METHOD Execute : HRESULT
VAR_INST
	_GetEventState	: UINT; // Step variable
	_BufferOverflow : BOOL; // Buffer maximum reached
END_VAR

VAR
	_TmpAlarm : Tc3_PackML_V2.ST_Alarm; // temp. Alarm structure
	_hr		  : HRESULT;				// HResult
END_VAR
IF __ISVALIDREF(_AdminTag) THEN
	IF _InternalErrorAck AND _InternalError THEN
		_InternalError := FALSE;
	END_IF

	IF _InternalError THEN
		RETURN;
	END_IF

	IF THIS^.GetTimeZone THEN
		IF THIS^.TimeZone() THEN
			THIS^.GetTimeZone := FALSE;
		END_IF
	END_IF

	IF NOT THIS^.GetTimeZone AND THIS^.EventsSubscribed THEN
		Execute := SUPER^.Execute(); // retrieve events
		CASE _GetEventState OF
			0: // Idle
				IF CntAlarmsRaised > 0 THEN
					THIS^.NewEvent := FALSE;
					_GetEventState := _GetEventState + 1;
				END_IF

			1: // handle the event		
				IF aEventInfoBuffer[CntAlarmsRaised].fbRequestEventText.bError THEN
					Tc2_System.ADSLOGSTR(msgCtrlMask := cMsgCtrlMask, msgFmtStr := Tc2_Standard.CONCAT(cBaseMsg, 'Execute: %s'), strArg := 'REQUEST EVENTTEXT ERROR');
					_GetEventState := 0;
					_InternalError := TRUE;
				ELSIF NOT aEventInfoBuffer[CntAlarmsRaised].fbRequestEventText.bBusy THEN
					aEventInfoBuffer[CntAlarmsRaised].fbRequestEventText.GetString(aEventInfoBuffer[CntAlarmsRaised].EventText, SIZEOF(Tc3_PackML_V2.ST_Alarm.Message));
					_hr := THIS^.WriteAlarmTags(Alarm_Ref	  := _TmpAlarm,
												EventInfo_Ref := THIS^.aEventInfoBuffer[CntAlarmsRaised],
												Trigger		  := TRUE,
												AlarmIndex	  := CntAlarmsRaised);

					IF Tc3_Module.SUCCEEDED(_hr) THEN
						// Critical / StopReason 
						IF THIS^.aEventInfoBuffer[CntAlarmsRaised].eSeverity = TcEventSeverity.Critical THEN // Check "Critical" --> Stop reason
							_hr := THIS^.AlarmArrayHandler(NewAlarm_Ref			:= _TmpAlarm,
														   ActAlarmsCounter_Ref := UnclearedStopReasons,
														   MaxArrayElements		:= Tc3_PackML_V2.MaxStopReasons,
														   pAlarmArray			:= ADR(_AdminTag.StopReason),
														   BufferOverflow_Ref	:= _BufferOverflow);

							IF _BufferOverflow THEN
								Tc2_System.ADSLOGSTR(msgCtrlMask := Tc2_System.ADSLOG_MSGTYPE_ERROR, msgFmtStr := Tc2_Standard.CONCAT(cBaseMsg, 'Execute: %s'), strArg := 'Stop reason Buffer is full / FIFO active');
								_BufferOverflow := FALSE;
							END_IF

						// Alarm (StopReason) 
						ELSIF THIS^.aEventInfoBuffer[CntAlarmsRaised].eSeverity = TcEventSeverity.Error THEN // Check "Error" --> Alarm

							// Alarm handling
							_hr := THIS^.AlarmArrayHandler(NewAlarm_Ref			:= _TmpAlarm,
														   ActAlarmsCounter_Ref := UnclearedAlarms,
														   MaxArrayElements		:= Tc3_PackML_V2.MaxAlarms,
														   pAlarmArray			:= ADR(_AdminTag.Alarm),
														   BufferOverflow_Ref	:= _BufferOverflow);

							IF _BufferOverflow THEN
								Tc2_System.ADSLOGSTR(msgCtrlMask := Tc2_System.ADSLOG_MSGTYPE_ERROR, msgFmtStr := Tc2_Standard.CONCAT(cBaseMsg, 'Execute: %s'), strArg := 'Alarm Buffer is full / FIFO active');
								_BufferOverflow := FALSE;
							END_IF

							// to StopReason
							IF _AlarmToStopReason AND Tc3_Module.SUCCEEDED(_hr) THEN
								_hr := THIS^.AlarmArrayHandler(NewAlarm_Ref			:= _TmpAlarm,
															   ActAlarmsCounter_Ref := UnclearedStopReasons,
															   MaxArrayElements		:= Tc3_PackML_V2.MaxStopReasons,
															   pAlarmArray			:= ADR(_AdminTag.StopReason),
															   BufferOverflow_Ref	:= _BufferOverflow);

								IF _BufferOverflow THEN
									Tc2_System.ADSLOGSTR(msgCtrlMask := Tc2_System.ADSLOG_MSGTYPE_ERROR, msgFmtStr := Tc2_Standard.CONCAT(cBaseMsg, 'Execute: %s'), strArg := 'Stop reason Buffer is full / FIFO active');
									_BufferOverflow := FALSE;
								END_IF
							END_IF
						// Warning (StopReason) 
						ELSIF THIS^.aEventInfoBuffer[CntAlarmsRaised].eSeverity = TcEventSeverity.Warning THEN // Check "Warning" --> Warning
							_hr := THIS^.AlarmArrayHandler(NewAlarm_Ref			:= _TmpAlarm,
														   ActAlarmsCounter_Ref := UnclearedWarnings,
														   MaxArrayElements		:= Tc3_PackML_V2.MaxWarnings,
														   pAlarmArray			:= ADR(_AdminTag.Warning),
														   BufferOverflow_Ref	:= _BufferOverflow);

							IF _BufferOverflow THEN
								Tc2_System.ADSLOGSTR(msgCtrlMask := Tc2_System.ADSLOG_MSGTYPE_ERROR, msgFmtStr := Tc2_Standard.CONCAT(cBaseMsg, 'Execute: %s'), strArg := 'Warning Buffer is full / FIFO active');
								_BufferOverflow := FALSE;
							END_IF

							// to StopReason
							IF _WarningToStopReason AND Tc3_Module.SUCCEEDED(_hr) THEN
								_hr := THIS^.AlarmArrayHandler(NewAlarm_Ref			:= _TmpAlarm,
															   ActAlarmsCounter_Ref := UnclearedStopReasons,
															   MaxArrayElements		:= Tc3_PackML_V2.MaxStopReasons,
															   pAlarmArray			:= ADR(_AdminTag.StopReason),
															   BufferOverflow_Ref	:= _BufferOverflow);

								IF _BufferOverflow THEN
									Tc2_System.ADSLOGSTR(msgCtrlMask := Tc2_System.ADSLOG_MSGTYPE_ERROR, msgFmtStr := Tc2_Standard.CONCAT(cBaseMsg, 'Execute: %s'), strArg := 'Stop reason Buffer is full / FIFO active');
									_BufferOverflow := FALSE;
								END_IF
							END_IF
						END_IF

						IF Tc3_Module.SUCCEEDED(_hr) THEN
							CntAlarmsRaised := CntAlarmsRaised - 1;
							_GetEventState	:= 0;
						END_IF
					END_IF
				END_IF

		ELSE
			Tc2_System.ADSLOGSTR(msgCtrlMask := cMsgCtrlMask, msgFmtStr := Tc2_Standard.CONCAT(cBaseMsg, 'Execute: %s'), strArg := 'Case Idx error');
			_InternalError := TRUE;
		END_CASE

		THIS^.GetMsgInfos();
	END_IF
ELSE
	IF NOT _InternalError THEN
		// Set internal Error
		Tc2_System.ADSLOGSTR(msgCtrlMask := cMsgCtrlMask, msgFmtStr := Tc2_Standard.CONCAT(cBaseMsg, 'Execute: %s'), strArg := 'Input-reference error');
		_InternalError := TRUE;
	END_IF
END_IF
END_METHOD

METHOD PUBLIC GetMsgInfos : ST_PackML_aEventInfo
VAR
	_Iterator : DINT; // FOR-Loop iterator						
END_VAR
// StopReason

// Reset
GetMsgInfos.StopReason.Active		   := FALSE;
GetMsgInfos.StopReason.NumberActive	   := 0;
GetMsgInfos.StopReason.NumberConfirmed := 0;
GetMsgInfos.StopReason.NumberCleared   := 0;
FOR _Iterator := 1 TO Tc3_PackML_V2.MaxStopReasons DO
	// Active
	IF _AdminTag.StopReason[_Iterator].Trigger THEN
		GetMsgInfos.StopReason.Active		:= TRUE;
		GetMsgInfos.StopReason.NumberActive := GetMsgInfos.StopReason.NumberActive + 1;
	END_IF

	// Confirmed
	IF NOT _AdminTag.StopReason[_Iterator].Trigger AND (_AdminTag.StopReason[_Iterator].Category = 4) THEN
		GetMsgInfos.StopReason.NumberConfirmed := GetMsgInfos.StopReason.NumberConfirmed + 1;
	END_IF
END_FOR

// Alarm		

// Reset
GetMsgInfos.Alarm.Active		  := FALSE;
GetMsgInfos.Alarm.NumberActive	  := 0;
GetMsgInfos.Alarm.NumberConfirmed := 0;
GetMsgInfos.Alarm.NumberCleared	  := 0;
FOR _Iterator := 1 TO Tc3_PackML_V2.MaxAlarms DO
	// Active
	IF _AdminTag.Alarm[_Iterator].Trigger THEN
		GetMsgInfos.Alarm.Active	   := TRUE;
		GetMsgInfos.Alarm.NumberActive := GetMsgInfos.StopReason.NumberActive + 1;
	END_IF

	// Confirmed
	IF NOT _AdminTag.Alarm[_Iterator].Trigger AND (_AdminTag.Alarm[_Iterator].Category = 3) THEN
		GetMsgInfos.Alarm.NumberConfirmed := GetMsgInfos.Alarm.NumberConfirmed + 1;
	END_IF
END_FOR

// Warning		

// Reset
GetMsgInfos.Warning.Active			:= FALSE;
GetMsgInfos.Warning.NumberActive	:= 0;
GetMsgInfos.Warning.NumberConfirmed := 0;
GetMsgInfos.Warning.NumberCleared	:= 0;
FOR _Iterator := 1 TO Tc3_PackML_V2.MaxWarnings DO
	// Active
	IF _AdminTag.Warning[_Iterator].Trigger THEN
		GetMsgInfos.Warning.Active		 := TRUE;
		GetMsgInfos.Warning.NumberActive := GetMsgInfos.StopReason.NumberActive + 1;
	END_IF

	// Confirmed
	IF NOT _AdminTag.Warning[_Iterator].Trigger AND (_AdminTag.Warning[_Iterator].Category = 2) THEN
		GetMsgInfos.Warning.NumberConfirmed := GetMsgInfos.Warning.NumberConfirmed + 1;
	END_IF
END_FOR

// Cleared --> historizied
GetMsgInfos.HistorizedMsg := TO_UDINT(MsgInHistory);
FOR _Iterator := 1 TO Tc3_PackML_V2.MaxHistoryAlarms DO
	IF (_AdminTag.AlarmHistory[_Iterator].Category = 4) THEN // StopReason
		GetMsgInfos.StopReason.NumberCleared := GetMsgInfos.StopReason.NumberCleared + 1;
	ELSIF (_AdminTag.AlarmHistory[_Iterator].Category = 3) THEN // Alarm
		GetMsgInfos.Alarm.NumberCleared := GetMsgInfos.Alarm.NumberCleared + 1;
	ELSIF (_AdminTag.AlarmHistory[_Iterator].Category = 2) THEN // Warning
		GetMsgInfos.Warning.NumberCleared := GetMsgInfos.Warning.NumberCleared + 1;
	END_IF

	IF (_AdminTag.AlarmHistory[_Iterator].Category = 0) THEN
		EXIT;
	END_IF
END_FOR
END_METHOD

PROPERTY InitComplete : BOOL
GET
InitComplete := _InitComplete;
END_GET
END_PROPERTY

METHOD Initialize : BOOL
IF NOT EventsSubscribed THEN
	EventListener(Subscribe := TRUE, Subscribed => EventsSubscribed);
END_IF

Initialize := EventsSubscribed;
END_METHOD

PROPERTY InSimulation : BOOL
GET
InSimulation := _InSimulation;
END_GET
SET
_InSimulation := InSimulation;
END_SET
END_PROPERTY

PROPERTY InternalErrorAck : BOOL
GET
InternalErrorAck := _InternalErrorAck;
END_GET
SET
_InternalErrorAck := InternalErrorAck;
END_SET
END_PROPERTY

METHOD PRIVATE MoveAlarmToHistory : HRESULT
VAR_INPUT
	pAlarmArray		 : POINTER TO ST_Alarm; // Pointer to Array of ST_Alarm of Alarm / Warning / Stop reason
	ActAlarms_Ref	 : REFERENCE TO DINT;	// Reference to couter of active Alarm / Warning / Stop reason
	MaxArrayElements : INT;					// max. Alarm / Warning / Stop reason constant
	EventId			 : UDINT;				// EventId of Alarm / Warning / Stop reason to confirm
	Timestamp		 : ULINT;				// Event Timestamp
END_VAR

VAR
	_Iterator				  : INT;					// FOR-Loop iterator	
	_Iterator2				  : DINT;					// FOR-Loop iterator	
	_TempTimestruct			  : TIMESTRUCT;				// TimeStruct for ACK Time
	_TmpAlarm				  : Tc3_PackML_V2.ST_Alarm; // temp. Alarm Structure
	_hr						  : HRESULT;				// hresult
	_MaxArrayElementsInternal : INT;					// calculated internal Array upper border
	_BufferOverflow			  : BOOL;					// Buffer maximum reached
END_VAR
IF __ISVALIDREF(ActAlarms_Ref) THEN
	_MaxArrayElementsInternal := (MaxArrayElements - 1);

	// Search Alarm in Array
	FOR _Iterator := 0 TO _MaxArrayElementsInternal DO
		IF (pAlarmArray[_Iterator].ID = TO_DINT(EventId)) THEN
			// TimeZone
			THIS^.fbSpecificLocalTime(in := Tc2_Utilities.FILETIME64_TO_SYSTEMTIME(Timestamp), tzInfo := fbTimeZone.tzInfo, out => _TempTimestruct);

			// Copy Alarm to local Memory
			Tc2_System.MEMCPY(destAddr := ADR(_TmpAlarm), srcAddr := ADR(pAlarmArray[_Iterator]), n := SIZEOF(Tc3_PackML_V2.ST_Alarm));

			// Set ACK Timestamp	
			_TmpAlarm.AckDateTime[0] := TO_DINT(_TempTimestruct.wYear);
			_TmpAlarm.AckDateTime[1] := TO_DINT(_TempTimestruct.wMonth);
			_TmpAlarm.AckDateTime[2] := TO_DINT(_TempTimestruct.wDay);
			_TmpAlarm.AckDateTime[3] := TO_DINT(_TempTimestruct.wHour);
			_TmpAlarm.AckDateTime[4] := TO_DINT(_TempTimestruct.wMinute);
			_TmpAlarm.AckDateTime[5] := TO_DINT(_TempTimestruct.wSecond);
			_TmpAlarm.AckDateTime[6] := TO_DINT(_TempTimestruct.wMilliseconds);
			_TmpAlarm.Trigger		 := FALSE;

			// Move to History	
			_hr := THIS^.AlarmArrayHandler(NewAlarm_Ref			:= _TmpAlarm,
										   ActAlarmsCounter_Ref := THIS^.MsgInHistory,
										   MaxArrayElements		:= Tc3_PackML_V2.MaxHistoryAlarms,
										   pAlarmArray			:= ADR(_AdminTag.AlarmHistory),
										   BufferOverflow_Ref	:= _BufferOverflow);

			IF _BufferOverflow THEN
				Tc2_System.ADSLOGSTR(msgCtrlMask := Tc2_System.ADSLOG_MSGTYPE_ERROR, msgFmtStr := Tc2_Standard.CONCAT(cBaseMsg, 'MoveAlarmToHistory: %s'), strArg := 'History Buffer is full / FIFO active');
			END_IF

			IF Tc3_Module.SUCCEEDED(_hr) THEN
				// Close empty entry in source array
				Tc2_System.MEMMOVE(destAddr := ADR(pAlarmArray[_Iterator]), srcAddr := ADR(pAlarmArray[_Iterator + 1]), n := (SIZEOF(Tc3_PackML_V2.ST_Alarm) * (TO_UINT((_MaxArrayElementsInternal) - (_Iterator))))); // move Alarm 
				Tc2_System.MEMSET(destAddr := ADR(pAlarmArray[_MaxArrayElementsInternal]), fillByte := 0, n := SIZEOF(Tc3_PackML_V2.ST_Alarm));																		   // delete last entry

				// Find next empty entry index 
				FOR _Iterator2 := 0 TO (_MaxArrayElementsInternal) DO
					IF (pAlarmArray[_Iterator2].Message = '') OR (_Iterator2 = _MaxArrayElementsInternal) THEN
						IF _Iterator2 > 0 THEN
							ActAlarms_Ref := _Iterator2 - 1;
						ELSE
							ActAlarms_Ref := _Iterator2;
						END_IF

						EXIT;
					END_IF
				END_FOR
			END_IF

			EXIT;
		END_IF
	END_FOR

	MoveAlarmToHistory := S_OK;
ELSE
	// Set internal Error
	Tc2_System.ADSLOGSTR(msgCtrlMask := cMsgCtrlMask, msgFmtStr := Tc2_Standard.CONCAT(cBaseMsg, 'MoveAlarmToHistory: %s'), strArg := 'Input-reference error');
	MoveAlarmToHistory := E_FAIL;
	_InternalError	   := TRUE;
END_IF
END_METHOD

PROPERTY Name : STRING
GET
END_GET
SET
_Name := Name;
END_SET
END_PROPERTY

METHOD OnAlarmCleared : HRESULT
VAR_INPUT
	fbEvent : REFERENCE TO FB_TcEvent; // Reference to FB_Event (Callback!)
END_VAR

VAR_INST
	_idxEventReceived : INT; // Event index
END_VAR

VAR
	_hr : HRESULT; // hresult
END_VAR
// Move Alarm to History
IF fbEvent.eSeverity = TcEventSeverity.Critical THEN // Check "Critical" --> Stop reason
	_hr := MoveAlarmToHistory(MaxArrayElements := Tc3_PackML_V2.MaxStopReasons,
							  EventId		   := fbEvent.nEventId,
							  pAlarmArray	   := ADR(_AdminTag.StopReason),
							  Timestamp		   := fbEvent.nTimestamp,
							  ActAlarms_Ref	   := UnclearedStopReasons);
ELSIF fbEvent.eSeverity = TcEventSeverity.Error THEN // Check "Error" --> Alarm
	_hr := MoveAlarmToHistory(MaxArrayElements := Tc3_PackML_V2.MaxAlarms,
							  EventId		   := fbEvent.nEventId,
							  pAlarmArray	   := ADR(_AdminTag.Alarm),
							  Timestamp		   := fbEvent.nTimestamp,
							  ActAlarms_Ref	   := UnclearedAlarms);

	IF _AlarmToStopReason AND Tc3_Module.SUCCEEDED(_hr) THEN
		_hr := THIS^.ClearStopReason(pAlarmArray	  := ADR(_AdminTag.StopReason),
									 ActAlarms_Ref	  := THIS^.UnclearedStopReasons,
									 MaxArrayElements := Tc3_PackML_V2.MaxStopReasons,
									 EventId		  := fbEvent.nEventId);
	END_IF
ELSIF fbEvent.eSeverity = TcEventSeverity.Warning THEN // Check "Warning" --> Warning
	_hr := MoveAlarmToHistory(MaxArrayElements := Tc3_PackML_V2.MaxWarnings,
							  EventId		   := fbEvent.nEventId,
							  pAlarmArray	   := ADR(_AdminTag.Warning),
							  Timestamp		   := fbEvent.nTimestamp,
							  ActAlarms_Ref	   := UnclearedWarnings);

	IF _WarningToStopReason AND Tc3_Module.SUCCEEDED(_hr) THEN
		_hr := THIS^.ClearStopReason(pAlarmArray	  := ADR(_AdminTag.StopReason),
									 ActAlarms_Ref	  := THIS^.UnclearedStopReasons,
									 MaxArrayElements := Tc3_PackML_V2.MaxStopReasons,
									 EventId		  := fbEvent.nEventId);
	END_IF
END_IF

OnAlarmCleared := S_OK; // in order to receive more callbacks (Set <> S_OK in order to cancel the callbacks for this program cycle.)
END_METHOD

// Callback Method
METHOD OnAlarmConfirmed : HRESULT
VAR_INPUT
	fbEvent : REFERENCE TO FB_TcEvent; // Reference to FB_Event (Callback!)
END_VAR

VAR
	_hr : HRESULT; // hresult
END_VAR
// Move Alarm to History
IF __ISVALIDREF(fbEvent) THEN
	// Set ACK Timestamp
	IF fbEvent.eSeverity = TcEventSeverity.Critical THEN // Check "Critical" --> Stop reason
		_hr := ConfirmAlarm(MaxArrayElements := Tc3_PackML_V2.MaxStopReasons,
							EventId			 := fbEvent.nEventId,
							pAlarmArray		 := ADR(_AdminTag.StopReason),
							Timestamp		 := fbEvent.nTimestamp,
							ActAlarms_Ref	 := UnclearedStopReasons);
	ELSIF fbEvent.eSeverity = TcEventSeverity.Error THEN // Check "Error" --> Alarm
		_hr := ConfirmAlarm(MaxArrayElements := Tc3_PackML_V2.MaxAlarms,
							EventId			 := fbEvent.nEventId,
							pAlarmArray		 := ADR(_AdminTag.Alarm),
							Timestamp		 := fbEvent.nTimestamp,
							ActAlarms_Ref	 := UnclearedAlarms);
	ELSIF fbEvent.eSeverity = TcEventSeverity.Warning THEN // Check "Warning" --> Warning
		_hr := ConfirmAlarm(MaxArrayElements := Tc3_PackML_V2.MaxWarnings,
							EventId			 := fbEvent.nEventId,
							pAlarmArray		 := ADR(_AdminTag.Warning),
							Timestamp		 := fbEvent.nTimestamp,
							ActAlarms_Ref	 := UnclearedWarnings);
	END_IF

	OnAlarmConfirmed := S_OK; // in order to receive more callbacks (Set <> S_OK in order to cancel the callbacks for this program cycle.)
ELSE
	// Set internal Error
	Tc2_System.ADSLOGSTR(msgCtrlMask := cMsgCtrlMask, msgFmtStr := Tc2_Standard.CONCAT(cBaseMsg, 'OnAlarmConfirmed: %s'), strArg := 'Input-reference error');
	OnAlarmConfirmed := E_FAIL;
	_InternalError	 := TRUE;
END_IF
END_METHOD

// Callback Method
METHOD OnAlarmRaised : HRESULT
VAR_INPUT
	fbEvent : REFERENCE TO FB_TcEvent; // Reference to FB_Event (Callback!)
END_VAR

VAR
	_TempTimestruct : TIMESTRUCT; // TimeStruct for ACK Time
END_VAR
// when (new) event is triggered -> trigger within cyclic method 'execute'
THIS^.NewEvent := TRUE;

// for local event -> raise counter
CntAlarmsRaised := CntAlarmsRaised + 1;

// save eventinfo locally
THIS^.stEventInfo.Source	  := fbEvent.ipSourceInfo.sName;
THIS^.stEventInfo.eSeverity	  := fbEvent.eSeverity;
THIS^.stEventInfo.EventClass  := fbEvent.EventClass;
THIS^.stEventInfo.EventId	  := fbEvent.nEventId;
THIS^.stEventInfo.ipArguments := fbEvent.ipArguments;

// TimeZone
fbSpecificLocalTime(in := Tc2_Utilities.FILETIME64_TO_SYSTEMTIME(fbEvent.nTimestamp), tzInfo := fbTimeZone.tzInfo, out => _TempTimestruct);

// Timestamp	
THIS^.stEventInfo.TimeRaised[0] := TO_DINT(_TempTimestruct.wYear);
THIS^.stEventInfo.TimeRaised[1] := TO_DINT(_TempTimestruct.wMonth);
THIS^.stEventInfo.TimeRaised[2] := TO_DINT(_TempTimestruct.wDay);
THIS^.stEventInfo.TimeRaised[3] := TO_DINT(_TempTimestruct.wHour);
THIS^.stEventInfo.TimeRaised[4] := TO_DINT(_TempTimestruct.wMinute);
THIS^.stEventInfo.TimeRaised[5] := TO_DINT(_TempTimestruct.wSecond);
THIS^.stEventInfo.TimeRaised[6] := TO_DINT(_TempTimestruct.wMilliseconds);
Tc2_System.MEMSET(destAddr := ADR(stEventInfo.TimeCleared), fillByte := 0, n := SIZEOF(stEventInfo.TimeCleared));
Tc2_System.MEMSET(destAddr := ADR(stEventInfo.TimeConfirmed), fillByte := 0, n := SIZEOF(stEventInfo.TimeConfirmed));

// store event info globally
aEventInfoBuffer[CntAlarmsRaised] := stEventInfo;

// activate requests in event triggered method 'OnMessageSent' to get related request info
aEventInfoBuffer[CntAlarmsRaised].fbRequestEventText.Request(eventClass := aEventInfoBuffer[CntAlarmsRaised].EventClass,
															 nEventId	:= aEventInfoBuffer[CntAlarmsRaised].EventId,
															 nLangId	:= 1033,
															 ipArgs		:= aEventInfoBuffer[CntAlarmsRaised].ipArguments);

OnAlarmRaised := S_OK; // in order to receive more callbacks (Set <> S_OK in order to cancel the callbacks for this program cycle.)
END_METHOD

PROPERTY ParentResponseDefinitions : ARRAY[0..4] OF SPT_BaseTypes.E_AlarmResponse
GET
ParentResponseDefinitions := _ParentResponseDefinitions;
END_GET
SET
_ParentResponseDefinitions := ParentResponseDefinitions;
END_SET
END_PROPERTY

METHOD Reset : BOOL
// This may or may not be called depending on the component type 

// which derives FB_ComponentBase
F_ClearAllEventsInClass(PackMLEventHandlerAlarms);
Reset := TRUE;
END_METHOD

METHOD PUBLIC TimeZone : BOOL
VAR_INST
	_Step : USINT; // Step Variable
END_VAR
CASE _Step OF
	0: // Start to get local Timezone 
		fbTimeZone.bExecute := TRUE;
		IF fbTimeZone.bBusy THEN
			_Step := _Step + 1;
		END_IF

	1: // set 
		fbTimeZone.bExecute := FALSE;
		_Step				:= 0;
		TimeZone			:= TRUE;

ELSE
	Tc2_System.ADSLOGSTR(msgCtrlMask := cMsgCtrlMask, msgFmtStr := Tc2_Standard.CONCAT(cBaseMsg, 'TimeZone: %s'), strArg := 'Case Idx error');
	_InternalError := TRUE;
END_CASE

fbTimeZone(sNetID := '');
IF fbTimeZone.bError THEN
	Tc2_System.ADSLOGSTR(msgCtrlMask := cMsgCtrlMask, msgFmtStr := Tc2_Standard.CONCAT(cBaseMsg, 'fbTimeZone ErrID: %s'), strArg := TO_STRING(fbTimeZone.nErrID));
	_InternalError := TRUE;
END_IF
END_METHOD

PROPERTY WarningToStopReason : BOOL
SET
_WarningToStopReason := WarningToStopReason;
END_SET
END_PROPERTY

METHOD PRIVATE WriteAlarmTags : HRESULT;
VAR_INPUT
	Alarm_Ref	  : REFERENCE TO Tc3_PackML_V2.ST_Alarm; // Reference to ST_Alarm of an new Alarm / Warning / Stop reason
	EventInfo_Ref : REFERENCE TO ST_EventInfo;			 // Reference to ST_EventInfo
	Trigger		  : BOOL;								 // Set / Reset Trigger in PML Structure
	AlarmIndex	  : DINT;								 // Alarm index
END_VAR
IF __ISVALIDREF(Alarm_Ref) AND __ISVALIDREF(EventInfo_Ref) THEN
	Alarm_Ref.ID	   := TO_DINT(EventInfo_Ref.EventId);
	Alarm_Ref.Value	   := AlarmIndex;
	Alarm_Ref.Message  := EventInfo_Ref.EventText;
	Alarm_Ref.Category := TO_DINT(EventInfo_Ref.eSeverity); // Verbose:=0, Info:=1, Warning:=2, Error:=3, Critical:=4
	Alarm_Ref.Trigger  := Trigger;
	Alarm_Ref.DateTime := EventInfo_Ref.TimeRaised;
	WriteAlarmTags	   := S_OK;
ELSE
	// Set internal Error
	Tc2_System.ADSLOGSTR(msgCtrlMask := cMsgCtrlMask, msgFmtStr := Tc2_Standard.CONCAT(cBaseMsg, 'WriteAlarmTags: %s'), strArg := 'Input-reference error');
	WriteAlarmTags := E_FAIL;
	_InternalError := TRUE;
END_IF
END_METHOD

END_FUNCTION_BLOCK

// Project Information/F_GetCompany
// This function has been automatically generated from the project information.
{attribute 'signature_flag' := '1073741824'}
{attribute 'TcGenerated'}
{attribute 'no-analysis'}
FUNCTION F_GetCompany : WSTRING
VAR_INPUT
	
END_VAR

F_GetCompany := "Beckhoff Automation LLC";

END_FUNCTION

// Project Information/F_GetTitle
// This function has been automatically generated from the project information.
{attribute 'signature_flag' := '1073741824'}
{attribute 'TcGenerated'}
{attribute 'no-analysis'}
FUNCTION F_GetTitle : WSTRING
VAR_INPUT
	
END_VAR

F_GetTitle := "SPT Components";

END_FUNCTION

// Project Information/F_GetVersion
// This function has been automatically generated from the project information.
{attribute 'signature_flag' := '1073741824'}
{attribute 'TcGenerated'}
{attribute 'no-analysis'}
FUNCTION F_GetVersion : ST_LibVersion
VAR_INPUT
	
END_VAR

F_GetVersion.iMajor := 3;
F_GetVersion.iMinor := 9;
F_GetVersion.iBuild := 0;
F_GetVersion.iRevision := 0;
F_GetVersion.sVersion := '3.9.0';
F_GetVersion.nFlags := 1;

END_FUNCTION

// Sensors/FB_DigitalSensor
FUNCTION_BLOCK FB_DigitalSensor EXTENDS FB_ComponentBase IMPLEMENTS I_DigitalSensorBase
VAR
	HardwareInput AT %I*		: BOOL;			  // Hardware input bit from the physical sensor
	_DebounceMode				: E_DebounceMode; // Defines the debounce model that will filter the sensor's output to the program
	_DebounceTime				: TIME;			  // Time input parameter for use in Debounce functionality
	_Inverted					: BOOL;			  // Defines the output polarity of the sensor - a "TRUE" value will result in the signal of the sensor being inverted
	_SimulationInput			: BOOL;			  // Provides configuration input to the simulation functionality
	_SimulationTimebase			: UDINT;
	_SimulationMode				: E_SensorSimulationMode; // Defines the mode of operation for the simulation functionality of this component
	_TimeActive					: TIME;					  // Tracks the amount of time that the sensor has been in an active state
	_TimeInactive				: TIME;					  // Tracks the amount of time that the sensor has been in an inactive state
	_Active						: BOOL;
	TON_ActiveTimer				: Tc2_Standard.TON; // Tracks the amount of time that the sensor has been in an active state
	TON_InactiveTimer			: Tc2_Standard.TON; // Tracks the amount of time that the sensor has been in an inactive state
	TON_DebounceTimer			: Tc2_Standard.TON; // Utilized in the debounce implementation
	TP_DebounceTimer			: Tc2_Standard.TP;	// Utilized in the debounce implementation
	DigitalSensor_HMI			: ST_DigitalSensor_HMI;
	SimulationPulse1_TP			: Tc2_Standard.TP; // Pulse Timer for simulated sensor pulse generation
	SimulationPulse2_TP			: Tc2_Standard.TP; // Pulse Timer for simulated sensor pulse generation
	HMICommand_DigitalSensor_RT : R_TRIG;
END_VAR

METHOD PUBLIC CyclicLogic
VAR_INPUT
END_VAR
SUPER^.CyclicLogic();
IF _Simulate THEN
	CASE _SimulationMode OF
		E_SensorSimulationMode.InputDriven:
			_Active := _SimulationInput;

		E_SensorSimulationMode.Periodic:
			SimulationPulse1_TP(IN := NOT SimulationPulse2_TP.Q, PT := UDINT_TO_TIME(_SimulationTimebase));
			SimulationPulse2_TP(IN := NOT SimulationPulse1_TP.Q, PT := UDINT_TO_TIME(_SimulationTimebase));
			_Active := SimulationPulse2_TP.Q;
	END_CASE
ELSE
	_Active := ProcessInput(Input := HardwareInput);
END_IF
END_METHOD

PROPERTY Active : BOOL
GET
Active := _Active;
END_GET
END_PROPERTY

PROPERTY DebounceMode : E_DebounceMode
GET
DebounceMode := _DebounceMode;
END_GET
SET
_DebounceMode := DebounceMode;
END_SET
END_PROPERTY

PROPERTY DebounceTime : TIME
GET
DebounceTime := _DebounceTime;
END_GET
SET
_DebounceTime := DebounceTime;
END_SET
END_PROPERTY

PROPERTY Inverted : BOOL
GET
Inverted := _Inverted;
END_GET
SET
_Inverted := Inverted;
END_SET
END_PROPERTY

PROPERTY SimulationInput : BOOL
GET
SimulationInput := _SimulationInput;
END_GET
SET
_SimulationInput := SimulationInput;
END_SET
END_PROPERTY

PROPERTY SimulationMode : E_SensorSimulationMode
GET
SimulationMode := _SimulationMode;
END_GET
SET
_SimulationMode := SimulationMode;
END_SET
END_PROPERTY

PROPERTY SimulationTimeBase : UDINT
GET
SimulationTimeBase := _SimulationTimebase;
END_GET
SET
_SimulationTimeBase := SimulationTimebase;
END_SET
END_PROPERTY

PROPERTY TimeActive : TIME
GET
TimeActive := _TimeActive;
END_GET
END_PROPERTY

PROPERTY TimeInactive : TIME
GET
TimeInactive := _TimeInactive;
END_GET
END_PROPERTY

METHOD PROTECTED HMICommunication
// Extend this method in extended FBs to communicate specific implementation data
SUPER^.HMICommunication();

// Process HMI requests

// Replace 'FALSE' below with further momentary commands (myCommand XOR myOtherCommand XOR...)
HMICommand_DigitalSensor_RT(CLK := (ComponentBase_HMI.Status.HMIControlAvailable AND NOT HMICommandActive_Base) AND (FALSE));

// Signal to FB_ComponentBase that a command is active
HMICommandActive_Descendant := ComponentBase_HMI.Status.HMIControlAvailable AND (DigitalSensor_HMI.Config.DebounceMode <> _DebounceMode OR DigitalSensor_HMI.Config.DebounceTime <> _DebounceTime OR DigitalSensor_HMI.Config.Inverted <> _Inverted OR DigitalSensor_HMI.Config.SimulationMode <> _SimulationMode OR DigitalSensor_HMI.Config.SimulationTimebase <> _SimulationTimebase);

// Process HMI requests
IF HMICommand_DigitalSensor_RT.Q THEN // If a request has been issued by the HMI, and a previous request has not just finished being processed

	//	IF AxisBaseHMI.Command.xxx THEN

	//		Enabled := TRUE;

	//	END_IF
END_IF

IF ComponentBase_HMI.Status.HMIControlAvailable AND NOT HMICommand_DigitalSensor_RT.Q THEN
	IF DigitalSensor_HMI.Config.DebounceMode <> _DebounceMode THEN
		DebounceMode := DigitalSensor_HMI.Config.DebounceMode;
	END_IF

	IF DigitalSensor_HMI.Config.DebounceTime <> _DebounceTime THEN
		DebounceTime := DigitalSensor_HMI.Config.DebounceTime;
	END_IF

	IF DigitalSensor_HMI.Config.Inverted <> _Inverted THEN
		Inverted := DigitalSensor_HMI.Config.Inverted;
	END_IF

	IF DigitalSensor_HMI.Config.SimulationMode <> _SimulationMode THEN
		SimulationMode := DigitalSensor_HMI.Config.SimulationMode;
	END_IF

	IF DigitalSensor_HMI.Config.SimulationTimebase <> _SimulationTimebase THEN
		SimulationTimeBase := DigitalSensor_HMI.Config.SimulationTimebase;
	END_IF
END_IF

// Update HMI status info
DigitalSensor_HMI.Status.Active				:= _Active;
DigitalSensor_HMI.Status.TimeActive			:= TIME_TO_LREAL(_TimeActive) / 1000.0;
DigitalSensor_HMI.Status.TimeInactive		:= TIME_TO_LREAL(_TimeInactive) / 1000.0;
DigitalSensor_HMI.Config.DebounceMode		:= DebounceMode;
DigitalSensor_HMI.Config.DebounceTime		:= DebounceTime;
DigitalSensor_HMI.Config.Inverted			:= Inverted;
DigitalSensor_HMI.Config.SimulationMode		:= SimulationMode;
DigitalSensor_HMI.Config.SimulationTimebase := SimulationTimeBase;
END_METHOD

METHOD PROTECTED Monitoring
SUPER^.Monitoring();

// If flicker counters or other diagnostic systems are desired, their implementation could be here

// Any warnings, errors, or other desired messages would also be generated here

// T#71582M47S295MS is the upper bound of the TIME type, meaning these timers will continue to increase ET for as long as possible
TON_ActiveTimer(IN := _Active, PT := T#71582M47S295MS, ET => _TimeActive);
TON_InactiveTimer(IN := NOT _Active, PT := T#71582M47S295MS, ET => _TimeInactive);
_Busy  := FALSE;
_Error := FALSE;
END_METHOD

METHOD PRIVATE ProcessInput : BOOL
VAR_INPUT
	Input : BOOL;
END_VAR

VAR
	DebouncedInput : BOOL;
END_VAR

VAR_INST
	LastDebouncedInput : BOOL;
	MovingAverage	   : DINT;
END_VAR
CASE DebounceMode OF
	E_DebounceMode.RawInput: // Passes raw input through
		DebouncedInput := Input;

	E_DebounceMode.SimpleFlickerFilter:											 // Requires the raw input to be a consistent value for a set time period before output changes
		TON_DebounceTimer(IN := (Input <> DebouncedInput), PT := _DebounceTime); // runs the timer whenever a differing input is detected
		IF TON_DebounceTimer.Q THEN
			DebouncedInput := Input; // once the raw input has been different for the specified debounce time, the processed input is updated
		END_IF

	E_DebounceMode.EdgeDetectFilter:								   // Updates the processed value immediately on a change from steady state, but mutes any sensor flickers for the specified time immediately following the change
		IF (Input <> DebouncedInput) AND (NOT TP_DebounceTimer.Q) THEN // A differing raw input must be detected outside of the mute window created by the pulse timer
			DebouncedInput := Input;
		END_IF

		TP_DebounceTimer(IN := (DebouncedInput <> LastDebouncedInput), PT := _DebounceTime); // "Q" will be TRUE for tDebounce time after the bProcessedSensorInput value is changed
	E_DebounceMode.MovingAverage:															 // Uses a "moving average"-like calculation to compensate for extremely inconsistent signals - prevents poorly timed flickers from causing disproportionate results
		TON_DebounceTimer(IN := NOT TON_DebounceTimer.Q, PT := T#5MS);						 // Provides a 1ms "polling" trigger
		IF TON_DebounceTimer.Q THEN															 // TRUE once every millisecond
			IF Input THEN																	 // If raw input is currently active at the time of polling
				IF MovingAverage < TIME_TO_DINT(_DebounceTime) THEN							 // If the moving average has not reached its "weight limit" as set by debounce time
					MovingAverage := MovingAverage + 5;										 // Add 1 to the average
				END_IF
			ELSE													 // If raw input is currently inactive at the time of polling
				IF MovingAverage > -TIME_TO_DINT(_DebounceTime) THEN // If the moving average has not reached its "weight limit" as set by debounce time
					MovingAverage := MovingAverage - 5;				 // Subtract 1 from the average
				END_IF
			END_IF
		END_IF

		IF MovingAverage >= 0 THEN
			DebouncedInput := TRUE;
		ELSE
			DebouncedInput := FALSE;
		END_IF
END_CASE

LastDebouncedInput := DebouncedInput; // Update "Last value"
IF _Inverted THEN					  // If signal inversion is requested, invert the signal
	DebouncedInput := NOT DebouncedInput;
END_IF

ProcessInput := DebouncedInput;
END_METHOD

END_FUNCTION_BLOCK

// Sensors/I_DigitalSensorBase
INTERFACE I_DigitalSensorBase

PROPERTY Active : BOOL
GET
END_GET
END_PROPERTY

PROPERTY DebounceMode : E_DebounceMode
GET
END_GET
SET
END_SET
END_PROPERTY

PROPERTY DebounceTime : TIME
GET
END_GET
SET
END_SET
END_PROPERTY

PROPERTY Inverted : BOOL //"High" signal from the sensor will be interpreted as an "inactive" reading when this parameter is TRUE
GET
END_GET
SET
END_SET
END_PROPERTY

PROPERTY SimulationInput : BOOL
GET
END_GET
SET
END_SET
END_PROPERTY

PROPERTY SimulationMode : E_SensorSimulationMode
GET
END_GET
SET
END_SET
END_PROPERTY

PROPERTY TimeActive : TIME
GET
END_GET
END_PROPERTY

PROPERTY TimeInactive : TIME
GET
END_GET
END_PROPERTY

END_INTERFACE

// Solenoids/SolenoidBankBase/FB_SolenoidBankBase
FUNCTION_BLOCK ABSTRACT FB_SolenoidBankBase EXTENDS FB_ComponentBase
VAR
	// Configuration
	Configuration : ARRAY[1..Parameters_Cylinder.MAX_NUMBER_OF_SOLENOIDS] OF ST_SolenoidBankConfig;

	// Counted number of solenoids
	NumberOfSolenoids : UINT;

	// Alarms
	SolenoidBankAlarms : ARRAY[1..SolenoidBankBaseAlarmsCount] OF FB_TcAlarm;
END_VAR

VAR CONSTANT
	SolenoidBankBaseAlarmsCount : UINT := 2;
END_VAR

METHOD PUBLIC AddSolenoid : UINT
VAR_INPUT
	ipCylinder	 : I_Solenoid;
	Number		 : UINT; // This is the number in the IO tree.
	SolenoidType : E_SolenoidType;
END_VAR
IF CheckNumber(Number) AND ipCylinder <> 0 THEN
	NumberOfSolenoids									  := NumberOfSolenoids + 1;
	Configuration[NumberOfSolenoids].ipSolenoid			  := ipCylinder;
	Configuration[NumberOfSolenoids].SolenoidType		  := SolenoidType;
	Configuration[NumberOfSolenoids].SolenoidOutputNumber := Number;
END_IF
END_METHOD

METHOD PRIVATE CheckNumber : BOOL
VAR_INPUT
	Number : UINT;
END_VAR
CheckNumber := TRUE;
IF Number < 1 AND Number > Parameters_Cylinder.MAX_NUMBER_OF_SOLENOIDS THEN
	IF NOT SolenoidBankAlarms[E_CylinderBankAlarms.CylinderNumberOutOfRange].bRaised THEN
		SolenoidBankAlarms[E_CylinderBankAlarms.CylinderNumberOutOfRange].Raise(0);
	END_IF

	CheckNumber := FALSE;
END_IF
END_METHOD

METHOD PROTECTED CreateEvents
SUPER^.CreateEvents();
F_CreateAllEventsInClass(Alarms		:= SolenoidBankAlarms,
						 ClassSize	:= SIZEOF(TC_EVENTS.CylinderBankAlarms),
						 pInitEvent := ADR(TC_EVENTS.CylinderBankAlarms.InitReferenceEvent),
						 Prefix		:= Name);
END_METHOD

// This method serves as the entry point for all underlying FB logic
METHOD PUBLIC CyclicLogic
// This method should be called cyclically by descendant function blocks by invoking SUPER^.CyclicLogic().  Alternatively, the contents of this method could be reimplemented entirely in which case a call to this method would not be necessary.
VAR
	x : UINT;
END_VAR
// Loop through all solenoids that are added.
FOR x := 1 TO NumberOfSolenoids DO
	MapIO(x);
END_FOR
END_METHOD

// Basic component initialization logic
METHOD PROTECTED Initialize : BOOL;
// This method is called by CyclicLogic() as required
VAR
	x : UINT;
END_VAR
NumberOfSolenoids := 0;
Initialize		  := TRUE;
END_METHOD

METHOD ABSTRACT MapIO
VAR_INPUT
	x : UINT;
END_VAR
END_METHOD

// Provides basic error detection and event handling for this component
METHOD PROTECTED Monitoring

// This method is called cyclically by CyclicLogic()
SUPER^.Monitoring();
_CurrentAlarmSeverity := F_GetMaxSeverityRaised(Alarms := SolenoidBankAlarms, CurrentSeverity := CurrentAlarmSeverity);
END_METHOD

// Clears error flags and error IDs for this component
METHOD PUBLIC Reset : BOOL
SUPER^.Reset();
IF SolenoidBankAlarms[E_CylinderBankAlarms.CylinderNumberOutOfRange].bRaised THEN
	SolenoidBankAlarms[E_CylinderBankAlarms.CylinderNumberOutOfRange].Clear(0, 0);
END_IF
END_METHOD

END_FUNCTION_BLOCK

// Solenoids/I_Solenoid
INTERFACE I_Solenoid

METHOD Extend
VAR_INPUT
END_VAR
END_METHOD

PROPERTY Extended : BOOL
GET
END_GET
END_PROPERTY

PROPERTY ExtendOutput : BOOL
GET
END_GET
END_PROPERTY

PROPERTY ExtendTime : LREAL
GET
END_GET
SET
END_SET
END_PROPERTY

METHOD Retract
VAR_INPUT
END_VAR
END_METHOD

PROPERTY Retracted : BOOL
GET
END_GET
END_PROPERTY

PROPERTY RetractOutput : BOOL
GET
END_GET
END_PROPERTY

PROPERTY RetractTime : LREAL
GET
END_GET
SET
END_SET
END_PROPERTY

END_INTERFACE

// Solenoids/FB_DoubleSolenoid
FUNCTION_BLOCK FB_DoubleSolenoid EXTENDS FB_SingleSolenoid
VAR
	_RetractOutput AT %Q* : BOOL;
END_VAR

METHOD PROTECTED HardwareInit
// Update the status based on the IO 
IF _ExtendOutput AND NOT _RetractOutput THEN
	_Extended  := TRUE;
	_Retracted := FALSE;
ELSIF NOT _ExtendOutput AND _RetractOutput THEN
	_Extended  := FALSE;
	_Retracted := TRUE;
ELSE // By Default, set RetractOuptupt if neither is set or if both are set.
	_ExtendOutput  := FALSE;
	_RetractOutput := TRUE;
	_Extended	   := FALSE;
	_Retracted	   := TRUE;
END_IF
END_METHOD

METHOD PROTECTED HardwareUpdate
// One shot the requests
Extend_RTRIG(CLK := _ExtendRequest);
Retract_RTRIG(CLK := _RetractRequest);

// Handle Extend
IF Extend_RTRIG.Q THEN
	_ExtendOutput	:= TRUE;
	_RetractOutput	:= FALSE;
	_Extending		:= TRUE;
	_Retracting		:= FALSE;
	_Retracted		:= FALSE;
	_RetractRequest := FALSE;
END_IF

// Handle Retract
IF Retract_RTRIG.Q THEN
	_ExtendOutput  := FALSE;
	_RetractOutput := TRUE;
	_Extending	   := FALSE;
	_Retracting	   := TRUE;
	_Extended	   := FALSE;
	_ExtendRequest := FALSE;
END_IF

// Always Simulate Feedback here with no feedback inputs
Feedback();
END_METHOD

PROPERTY RetractOutput : BOOL
GET
RetractOutput := _RetractOutput;
END_GET
END_PROPERTY

END_FUNCTION_BLOCK

// Solenoids/FB_SingleSolenoid
(*	This FB is used for a single output solenoid 
	It uses the times to say when Extended/Retracted  	
	It starts assuming retracted and the output off.
*)
FUNCTION_BLOCK FB_SingleSolenoid EXTENDS FB_ComponentBase IMPLEMENTS I_Solenoid
VAR
	// Output
	_ExtendOutput AT %Q* : BOOL;

	// Internal variables
	_ExtendRequest	: BOOL;
	_RetractRequest : BOOL;
	_Extended		: BOOL;
	_Retracted		: BOOL;
	_Extending		: BOOL;
	_Retracting		: BOOL;
	_ExtendTime		: LREAL := 1000; // Default time 1s
	_RetractTime	: LREAL := 1000; // Default time 1s

	// Timer for Extend/Retract
	Extend_TON	  : TON;
	Retract_TON	  : TON;
	Extend_RTRIG  : R_TRIG;
	Retract_RTRIG : R_TRIG;

	// HMI 
	SolenoidHMI : ST_Cylinder_HMI;

	// Alarms
	SolenoidAlarms : ARRAY[1..SolenoidAlarmsCount] OF FB_TcAlarm;
END_VAR

VAR CONSTANT
	SolenoidAlarmsCount : UINT := 4;
END_VAR

METHOD PROTECTED CreateEvents
SUPER^.CreateEvents();
F_CreateAllEventsInClass(Alarms		:= SolenoidAlarms,
						 ClassSize	:= SIZEOF(TC_EVENTS.CylinderAlarms),
						 pInitEvent := ADR(TC_EVENTS.CylinderAlarms.InitReferenceEvent),
						 Prefix		:= Name);
END_METHOD

METHOD PROTECTED HMICommunication
VAR_INPUT
END_VAR
SUPER^.HMICommunication();

// Handle the requests to extend and retract
IF ComponentBase_HMI.Status.HMIControlAvailable THEN
	IF SolenoidHMI.Command.Extend THEN
		Extend();
	ELSIF SolenoidHMI.Command.Retract THEN
		Retract();
	END_IF

	IF NOT F_CompareLREAL(SolenoidHMI.Command.ExtendTime, _ExtendTime, 0.01) THEN
		_ExtendTime := SolenoidHMI.Command.ExtendTime;
	END_IF

	IF NOT F_CompareLREAL(SolenoidHMI.Command.RetractTime, _RetractTime, 0.01) THEN
		_RetractTime := SolenoidHMI.Command.RetractTime;
	END_IF
END_IF

// Update HMI status info
SolenoidHMI.Status.Extended	   := _Extended;
SolenoidHMI.Status.Extending   := _Extending;
SolenoidHMI.Status.Retracted   := _Retracted;
SolenoidHMI.Status.Retracting  := _Retracting;
SolenoidHMI.Config.ExtendTime  := _ExtendTime;
SolenoidHMI.Config.RetractTime := _RetractTime;
END_METHOD

METHOD PROTECTED Monitoring
VAR_INPUT
END_VAR
SUPER^.Monitoring();

// Update output bits
_Busy				  := _Extending OR _Retracting;
_CurrentAlarmSeverity := F_GetMaxSeverityRaised(Alarms := SolenoidAlarms, CurrentSeverity := CurrentAlarmSeverity);
_Error				  := _CurrentAlarmSeverity >= TcEventSeverity.Error;
END_METHOD

METHOD CyclicLogic
VAR
END_VAR
HardwareUpdate();
SUPER^.CyclicLogic();
END_METHOD

METHOD Extend
_ExtendRequest	:= TRUE;
_RetractRequest := FALSE;
END_METHOD

PROPERTY Extended : BOOL
GET
Extended := _Extended;
END_GET
END_PROPERTY

PROPERTY ExtendOutput : BOOL
GET
ExtendOutput := _ExtendOutput;
END_GET
END_PROPERTY

PROPERTY ExtendTime : LREAL
GET
ExtendTime := _ExtendTime;
END_GET
SET
_ExtendTime					   := ExtendTime;
SolenoidHMI.Command.ExtendTime := ExtendTime;
END_SET
END_PROPERTY

METHOD Retract
_ExtendRequest	:= FALSE;
_RetractRequest := TRUE;
END_METHOD

PROPERTY Retracted : BOOL
GET
Retracted := _Retracted;
END_GET
END_PROPERTY

PROPERTY RetractOutput : BOOL
GET
RetractOutput := FALSE;
END_GET
END_PROPERTY

PROPERTY RetractTime : LREAL
GET
RetractTime := _RetractTime;
END_GET
SET
_RetractTime					:= RetractTime;
SolenoidHMI.Command.RetractTime := RetractTime;
END_SET
END_PROPERTY

METHOD PROTECTED Feedback
VAR_INPUT
END_VAR
// Handle the time to Extend/Retract
Extend_TON(IN := _Extending, PT := LREAL_TO_TIME(_ExtendTime));
Retract_TON(IN := _Retracting, PT := LREAL_TO_TIME(_RetractTime));
IF Extend_TON.Q THEN
	_Extended  := TRUE;
	_Extending := FALSE;
END_IF

IF Retract_TON.Q THEN
	_Retracted	:= TRUE;
	_Retracting := FALSE;
END_IF
END_METHOD

METHOD PROTECTED HardwareInit
IF _ExtendOutput THEN
	_Extended  := TRUE;
	_Retracted := FALSE;
ELSE
	_Extended  := FALSE;
	_Retracted := TRUE;
END_IF
END_METHOD

METHOD PROTECTED HardwareUpdate
VAR_INPUT
END_VAR
// One shot the requests
Extend_RTRIG(CLK := _ExtendRequest);
Retract_RTRIG(CLK := _RetractRequest);

// Handle Extend
IF Extend_RTRIG.Q THEN
	_ExtendOutput	:= TRUE;
	_Extending		:= TRUE;
	_Retracting		:= FALSE;
	_Retracted		:= FALSE;
	_RetractRequest := FALSE;
END_IF

// Handle Retract
IF Retract_RTRIG.Q THEN
	_ExtendOutput  := FALSE;
	_Extending	   := FALSE;
	_Retracting	   := TRUE;
	_Extended	   := FALSE;
	_ExtendRequest := FALSE;
END_IF

// Call the feedback 
Feedback();
END_METHOD

// Basic component initialization logic
METHOD PROTECTED Initialize : BOOL;

// This method is called by CyclicLogic() as required
// Set the cylinder to retracted
_Extending		:= FALSE;
_ExtendRequest	:= FALSE;
_Retracting		:= FALSE;
_RetractRequest := FALSE;

// Set the HMI time to the currnt time.
SolenoidHMI.Command.ExtendTime	:= _ExtendTime;
SolenoidHMI.Command.RetractTime := _RetractTime;

// Call base class Initialize
Initialize := SUPER^.Initialize();

// Call the HardwareInit
HardwareInit();
END_METHOD

// Clears error flags and error IDs for this component
METHOD PUBLIC Reset : BOOL
SUPER^.Reset();
F_ClearAllEventsInClass(Alarms := SolenoidAlarms);
Reset := TRUE;
END_METHOD

END_FUNCTION_BLOCK

// Solenoids/FB_DoubleSolenoidFeedback
FUNCTION_BLOCK FB_DoubleSolenoidFeedback EXTENDS FB_DoubleSolenoid
VAR
	ExtendedSensor	AT %I* : BOOL;
	RetractedSensor AT %I* : BOOL;
END_VAR

PROPERTY ExtendedInput : BOOL
SET
ExtendedSensor := ExtendedInput;
END_SET
END_PROPERTY

METHOD PROTECTED Feedback
IF NOT _Simulate THEN
	_Extended  := ExtendedSensor;
	_Retracted := RetractedSensor;
	Extend_TON(IN := _Extending, PT := LREAL_TO_TIME(_ExtendTime));
	Retract_TON(IN := _Retracting, PT := LREAL_TO_TIME(_RetractTime));
	IF Extend_TON.Q AND NOT ExtendedSensor THEN
		IF NOT SolenoidAlarms[E_CylinderAlarms.ExtendTimeout].bRaised THEN
			SolenoidAlarms[E_CylinderAlarms.ExtendTimeout].Raise(0);
			_ExtendRequest := FALSE;
			_Extending	   := FALSE;
		END_IF
	ELSIF _Extending AND ExtendedSensor THEN
		_Extended  := TRUE;
		_Extending := FALSE;
	END_IF

	IF Retract_TON.Q AND NOT RetractedSensor THEN
		IF NOT SolenoidAlarms[E_CylinderAlarms.RetractTimeout].bRaised THEN
			SolenoidAlarms[E_CylinderAlarms.RetractTimeout].Raise(0);
			_RetractRequest := FALSE;
			_Retracting		:= FALSE;
		END_IF
	ELSIF _Retracting AND RetractedSensor THEN
		_Retracted	:= TRUE;
		_Retracting := FALSE;
	END_IF
ELSE
	SUPER^.Feedback();
END_IF

// Monitor Inputs in case both on at the same time
IF ExtendedSensor AND RetractedSensor AND NOT SolenoidAlarms[E_CylinderAlarms.ExtendedAndRetracted].bRaised THEN
	SolenoidAlarms[E_CylinderAlarms.ExtendedAndRetracted].Raise(0);
ELSIF (ExtendedSensor XOR RetractedSensor) AND SolenoidAlarms[E_CylinderAlarms.ExtendedAndRetracted].bRaised THEN
	SolenoidAlarms[E_CylinderAlarms.ExtendedAndRetracted].Clear(0, 0);
END_IF
END_METHOD

METHOD PROTECTED HardwareInit
IF ExtendedSensor AND NOT RetractedSensor THEN
	_Extended  := TRUE;
	_Retracted := FALSE;
ELSIF NOT ExtendedSensor AND RetractedSensor THEN
	_Extended  := FALSE;
	_Retracted := TRUE;
ELSE // With Neither on, then this means that it is not either or maybe no air
	_Extended  := FALSE;
	_Retracted := FALSE;
END_IF
END_METHOD

PROPERTY RetractedInput : BOOL
SET
RetractedSensor := RetractedInput;
END_SET
END_PROPERTY

END_FUNCTION_BLOCK

// Solenoids/FB_SingleSolenoidFeedback
FUNCTION_BLOCK FB_SingleSolenoidFeedback EXTENDS FB_SingleSolenoid
VAR
	ExtendedSensor	AT %I* : BOOL;
	RetractedSensor AT %I* : BOOL;
END_VAR

PROPERTY ExtendedInput : BOOL
SET
ExtendedSensor := ExtendedInput;
END_SET
END_PROPERTY

METHOD PROTECTED Feedback
IF NOT _Simulate THEN
	_Extended  := ExtendedSensor;
	_Retracted := RetractedSensor;
	Extend_TON(IN := _Extending, PT := LREAL_TO_TIME(_ExtendTime));
	Retract_TON(IN := _Retracting, PT := LREAL_TO_TIME(_RetractTime));
	IF Extend_TON.Q AND NOT ExtendedSensor THEN
		IF NOT SolenoidAlarms[E_CylinderAlarms.ExtendTimeout].bRaised THEN
			SolenoidAlarms[E_CylinderAlarms.ExtendTimeout].Raise(0);
			_ExtendRequest := FALSE;
			_Extending	   := FALSE;
		END_IF
	ELSIF _Extending AND ExtendedSensor THEN
		_Extended  := TRUE;
		_Extending := FALSE;
	END_IF

	IF Retract_TON.Q AND NOT RetractedSensor THEN
		IF NOT SolenoidAlarms[E_CylinderAlarms.RetractTimeout].bRaised THEN
			SolenoidAlarms[E_CylinderAlarms.RetractTimeout].Raise(0);
			_RetractRequest := FALSE;
			_Retracting		:= FALSE;
		END_IF
	ELSIF _Retracting AND RetractedSensor THEN
		_Retracted	:= TRUE;
		_Retracting := FALSE;
	END_IF
ELSE
	SUPER^.Feedback(); // Call the feedback that usese timers for feedback
END_IF

// Monitor Inputs in case both on at the same time
IF ExtendedSensor AND RetractedSensor AND NOT SolenoidAlarms[E_CylinderAlarms.ExtendedAndRetracted].bRaised THEN
	SolenoidAlarms[E_CylinderAlarms.ExtendedAndRetracted].Raise(0);
ELSIF (ExtendedSensor XOR RetractedSensor) AND SolenoidAlarms[E_CylinderAlarms.ExtendedAndRetracted].bRaised THEN
	SolenoidAlarms[E_CylinderAlarms.ExtendedAndRetracted].Clear(0, 0);
END_IF
END_METHOD

METHOD PROTECTED HardwareInit
IF ExtendedSensor AND NOT RetractedSensor THEN
	_Extended  := TRUE;
	_Retracted := FALSE;
ELSIF NOT ExtendedSensor AND RetractedSensor THEN
	_Extended  := FALSE;
	_Retracted := TRUE;
ELSE // With Neither on, then this means that it is not either or maybe no air
	_Extended  := FALSE;
	_Retracted := FALSE;
END_IF
END_METHOD

PROPERTY RetractedInput : BOOL
SET
RetractedSensor := RetractedInput;
END_SET
END_PROPERTY

END_FUNCTION_BLOCK
